FUNCTION_BLOCK OUT_BOOL (* Boolean Output Color Box *)
  (* Standard: 61499-1 *)
  (* Version 0.1, 2002-05-03, JHC, Rockwell Automation, Made QI IV=true. *)
  (* Version 0.0, 2001-04-14, JHC, Rockwell Automation, First XML version. *)
  (* Compiler header: package fb.rt.hmi; *)
  (* Compiler Java IBM VisualAge 3.0 *)
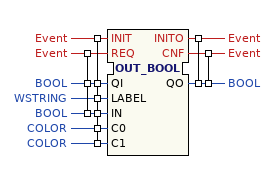
  EVENT_INPUT
    INIT WITH QI, LABEL, IN, C0, C1; (* Initialization *)
    REQ WITH QI, IN; (* Request *)
  END_EVENT
  EVENT_OUTPUT
    INITO WITH QO; (* Initialization Confirm *)
    CNF WITH QO; (* Service Confirmation *)
  END_EVENT
  VAR_INPUT
    QI : BOOL := true; (* Event qualifier *)
    LABEL : WSTRING; (* Label *)
    IN : BOOL; (* Input value *)
    C0 : COLOR := COLOR#white; (* Color when IN=0 *)
    C1 : COLOR := COLOR#green; (* Color when IN=1 *)
  END_VAR
  VAR_OUTPUT
    QO : BOOL; (* Event qualifier *)
  END_VAR
  FBS
    SEL : FB_SEL_COLOR;
    BOX : OUT_COLOR;
  END_FBS
  EVENT_CONNECTIONS
    INIT TO BOX.INIT;
    BOX.INITO TO INITO;
    REQ TO SEL.REQ;
    SEL.CNF TO BOX.REQ;
    BOX.CNF TO CNF;
  END_CONNECTIONS
  DATA_CONNECTIONS
    QI TO BOX.QI;
    BOX.QO TO QO;
    IN TO SEL.G;
    C0 TO SEL.IN0;
    C1 TO SEL.IN1;
    LABEL TO BOX.LABEL;
    SEL.OUT TO BOX.IN;
  END_CONNECTIONS
END_FUNCTION_BLOCK
